# B&R Automation Studio project Riesenrad_Noecker
Automation Studio 4.9

## Configuration Config1

### Hardware
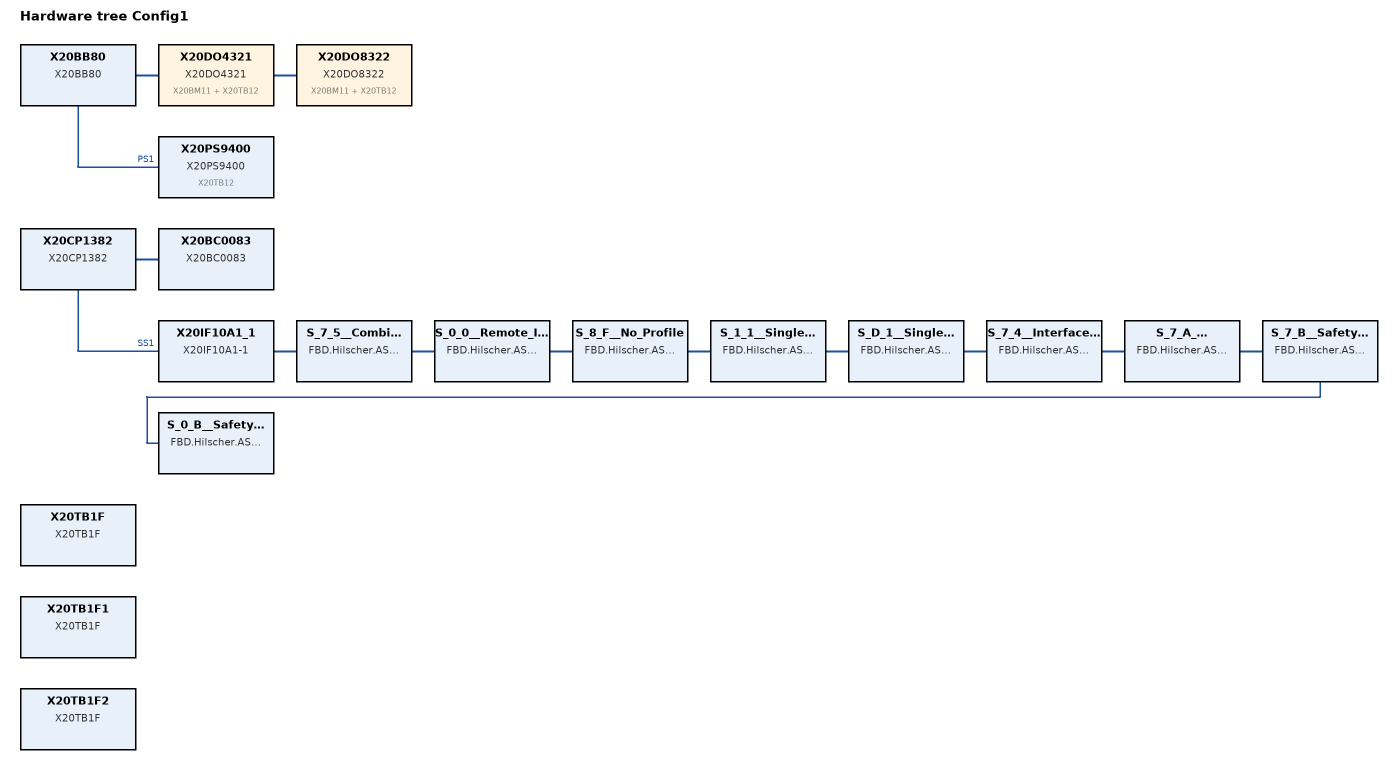
```
S_0_0__Remote_I_O_Port : FBD.Hilscher.AS-iSlaveDTM.S-0.0, Remote I$002FO Port vv.1 (OrderNumber=S-0.0, Remote I/O Port, VendorAddress=6)  [ASI1 -> S_7_5__Combi_field_device.ASI2]
  DtmId = cf450b26-e8ff-40bc-9c63-3c82782502b7
S_0_B__Safety_Slave : FBD.Hilscher.AS-iSlaveDTM.S-0.B, Safety Slave vv.1 (OrderNumber=S-0.B, Safety Slave, VendorAddress=13)  [ASI1 -> S_7_B__Safety_Slave.ASI2]
  DtmId = fa895fa4-d2e2-420c-b180-d2f2a02c2746
S_1_1__Single_Sensor__ext__contrl__ : FBD.Hilscher.AS-iSlaveDTM.S-1.1, Single Sensor (ext. contrl.) vv.1 (OrderNumber=S-1.1, Single Sensor (ext. contrl.), VendorAddress=8)  [ASI1 -> S_8_F__No_Profile.ASI2]
  DtmId = 9d5958e7-af56-4891-85b2-a17b108117c6
  ChannelBlocks_d3a35aad-8872-4e6a-914e-a881e2e31eaf  // Digital Input   [IN, 3 Bit(s)]
  ChannelBlocks_5bb377f7-42b1-4be2-805b-3354552dfad2  // Digital Output   [OUT, 1 Bit(s)]
S_7_4__Interface_for_16_bit_Signals : FBD.Hilscher.AS-iSlaveDTM.S-7.4, Interface for 16-bit Signals vv.1 (OrderNumber=S-7.4, Interface for 16-bit Signals, VendorAddress=10)  [ASI1 -> S_D_1__Single_Actuator_with_Monitoring.ASI2]
  DtmId = 0448b8e5-dced-4082-b80d-faf59c51bd2e
S_7_5__Combi_field_device : FBD.Hilscher.AS-iSlaveDTM.S-7.5, Combi field device vv.1 (OrderNumber=S-7.5, Combi field device, VendorAddress=5)  [ASI1 -> X20IF10A1_1.IF1]
  DtmId = 67ecf5d0-7b03-43bf-b517-437fc573c51f
S_7_A__Extended_Addressing_Mode : FBD.Hilscher.AS-iSlaveDTM.S-7.A, Extended Addressing Mode vv.1 (OrderNumber=S-7.A, Extended Addressing Mode, VendorAddress=11A)  [ASI1 -> S_7_4__Interface_for_16_bit_Signals.ASI2]
  DtmId = aa6d7d95-ba0b-4b78-a67e-6a7357710189
S_7_B__Safety_Slave : FBD.Hilscher.AS-iSlaveDTM.S-7.B, Safety Slave vv.1 (OrderNumber=S-7.B, Safety Slave, VendorAddress=12)  [ASI1 -> S_7_A__Extended_Addressing_Mode.ASI2]
  DtmId = 9a4111d3-a435-40ac-aa39-f4e884879d03
S_8_F__No_Profile : FBD.Hilscher.AS-iSlaveDTM.S-8.F, No Profile vv.1 (OrderNumber=S-8.F, No Profile, VendorAddress=7)  [ASI1 -> S_0_0__Remote_I_O_Port.ASI2]
  DtmId = 9c96085a-2bbf-4131-ae5e-8f64e9332ff0
S_D_1__Single_Actuator_with_Monitoring : FBD.Hilscher.AS-iSlaveDTM.S-D.1, Single Actuator with Monitoring vv.1 (OrderNumber=S-D.1, Single Actuator with Monitoring, VendorAddress=9)  [ASI1 -> S_1_1__Single_Sensor__ext__contrl__.ASI2]
  DtmId = 7ec07f93-a328-4a1d-a195-20a6fc18844a
  ChannelBlocks_4557325d-69fd-4a76-8f74-a661177b6065  // Digital Input   [IN, 3 Bit(s)]
  ChannelBlocks_a4a1c77a-8520-4756-9f44-c27872900355  // Digital Output   [OUT, 1 Bit(s)]
X20BB80 : X20BB80 v1.1.0.0
X20BC0083 : X20BC0083 v2.14.0.0  [PLK1 -> X20CP1382.IF3 (NodeNumber=1) [Cable Type=PowerlinkCable, Length=10, Version=1.0.0.3]; SL -> X20BB80.SL1]
X20BM11 : X20BM11 v1.1.0.0  [X2X1 -> X20BB80.IF1]
X20BM11a : X20BM11 v1.1.0.0  [X2X1 -> X20BM11.X2X2]
X20CP1382 : X20CP1382 v1.14.0.0  [X1 -> X1.SL; X2 -> X2.SL; X3 -> X3.SL]
  Module X1 (Type=X1, Virtual=true, Version=1.14.0.0)
    Connection (Connector=SS1, TargetModule=X20TB1F, TargetConnector=SS)
    Connection (Connector=SL, TargetModule=X20CP1382, TargetConnector=X1)
  Module X2 (Type=X2, Virtual=true, Version=1.14.0.0)
    Connection (Connector=SS1, TargetModule=X20TB1F1, TargetConnector=SS)
    Connection (Connector=SL, TargetModule=X20CP1382, TargetConnector=X2)
  Module X3 (Type=X3, Virtual=true, Version=1.14.0.0)
    Connection (Connector=SS1, TargetModule=X20TB1F2, TargetConnector=SS)
    Connection (Connector=SL, TargetModule=X20CP1382, TargetConnector=X3)
  Connector IF2:
    ActivateDevice = 1
    Mode = Manual
    InternetAddress = 192.168.0.10
    SubnetMask = 255.255.255.0
    ActivateSnmp = 2
  ConfigurationID = X20CP1382_Config1
  ActivateOpcUa = 1
  OpcUaInformationModels_PV_Version = 1
X20DO4321 : X20DO4321 v1.2.0.0  [SS1 -> X20TB12a.SS; SL -> X20BM11.SL1]
X20DO8322 : X20DO8322 v1.5.0.0  [SS1 -> X20TB12b.SS; SL -> X20BM11a.SL1]
X20IF10A1_1 : X20IF10A1-1 v1.3.0.0  [SS -> X20CP1382.SS1]
  Connector IF1:
    DtmId = c3d12960-2f64-4539-90e3-82e1d2b1aebe
  ConfigFile = X20IF10A1_1.dtm
  ConfigModule = asnxdb1
X20PS9400 : X20PS9400 v1.8.0.0  [SS1 -> X20TB12.SS; PS -> X20BB80.PS1]
X20TB12 : X20TB12 v1.0.0.0
X20TB12a : X20TB12 v1.0.0.0
X20TB12b : X20TB12 v1.0.0.0
X20TB1F : X20TB1F v1.0.0.0
X20TB1F1 : X20TB1F v1.0.0.0
X20TB1F2 : X20TB1F v1.0.0.0
```

### IoMap.iom - X20CP1382/IoMap.iom
```iecst
VAR_CONFIG
	::gDisplay AT %QW."S_7_5__Combi_field_device".Analog_Output_16_bit_Output_001;
	::gButtonOnOff AT %IX."S_0_0__Remote_I_O_Port".Digital_Input_1_bit_Input_001;
	::gButtonFast AT %IX."S_0_0__Remote_I_O_Port".Digital_Input_1_bit_Input_002;
	::gButtonSlow AT %IX."S_0_0__Remote_I_O_Port".Digital_Input_1_bit_Input_003;
	::gButtonStop AT %IX."S_0_0__Remote_I_O_Port".Digital_Input_1_bit_Input_004;
	::gRedDown AT %QX."S_8_F__No_Profile".Digital_Output_1_bit_Output_001;
	::gGreenDown AT %QX."S_8_F__No_Profile".Digital_Output_1_bit_Output_002;
	::gRedTop AT %QX."S_8_F__No_Profile".Digital_Output_1_bit_Output_003;
	::gGreenTop AT %QX."S_8_F__No_Profile".Digital_Output_1_bit_Output_004;
	::gReciever AT %IX."S_1_1__Single_Sensor__ext__contrl__".Digital_Input_1_bit_Input_001;
	::gTransmitter AT %QX."S_D_1__Single_Actuator_with_Monitoring".Digital_Output_1_bit_Output_001;
	::gRFIDColor AT %IW."S_7_4__Interface_for_16_bit_Signals".Analog_Input_16_bit_Input_001;
	::gASIStart AT %IX."S_7_A__Extended_Addressing_Mode".Digital_Input_1_bit_Input_001;
	::gASIStop AT %IX."S_7_A__Extended_Addressing_Mode".Digital_Input_1_bit_Input_002;
	::gASIQuit AT %IX."S_7_A__Extended_Addressing_Mode".Digital_Input_1_bit_Input_003;
	::gASISetup AT %IX."S_7_A__Extended_Addressing_Mode".Digital_Input_1_bit_Input_004;
	::gASILight1 AT %QX."S_7_A__Extended_Addressing_Mode".Digital_Output_1_bit_Output_001;
	::gASILight2 AT %QX."S_7_A__Extended_Addressing_Mode".Digital_Output_1_bit_Output_002;
	::gASILight3 AT %QX."S_7_A__Extended_Addressing_Mode".Digital_Output_1_bit_Output_003;
	::gEmergencyStop1 AT %IX."S_7_B__Safety_Slave".Digital_Input_1_bit_Input_001;
	::gEmergencyStop2 AT %IX."S_7_B__Safety_Slave".Digital_Input_1_bit_Input_002;
	::gEmergencyStop3 AT %IX."S_7_B__Safety_Slave".Digital_Input_1_bit_Input_003;
	::gEmergencyStop4 AT %IX."S_7_B__Safety_Slave".Digital_Input_1_bit_Input_004;
	::gLightGrid1 AT %IX."S_0_B__Safety_Slave".Digital_Input_1_bit_Input_001;
	::gLightGrid2 AT %IX."S_0_B__Safety_Slave".Digital_Input_1_bit_Input_002;
	::gLightGrid3 AT %IX."S_0_B__Safety_Slave".Digital_Input_1_bit_Input_003;
	::gLightGrid4 AT %IX."S_0_B__Safety_Slave".Digital_Input_1_bit_Input_004;
	::gDriveDirection AT %QX."X20DO4321".DigitalOutput01;
	::gDriveSpeed1 AT %QX."X20DO4321".DigitalOutput02;
	::gDriveSpeed2 AT %QX."X20DO4321".DigitalOutput03;
	::gSpotlightRight AT %QX."X20DO8322".DigitalOutput01;
	::gSpotlightLeft AT %QX."X20DO8322".DigitalOutput02;
	::gLightRed AT %QX."X20DO8322".DigitalOutput03;
	::gLightGreen AT %QX."X20DO8322".DigitalOutput04;
	::gLED1 AT %QX."X20DO8322".DigitalOutput05;
	::gLED2 AT %QX."X20DO8322".DigitalOutput06;
	::gLED3 AT %QX."X20DO8322".DigitalOutput07;
	::gLED4 AT %QX."X20DO8322".DigitalOutput08;
END_VAR
```

## Logical view

### Global.var - Globale Variablen
```iecst
(*List of global Variables*)
(* *)
VAR
	gSafetyStop : BOOL;
	gEmergencyStop : BOOL;
	gLightGrid : BOOL;
END_VAR
(*List of Variables for IO*)
(* *)
(*RFID*)
VAR
	gRFIDColor : UINT;
END_VAR
(* *)
(*Operating Light*)
VAR
	gRedTop : BOOL := FALSE;
	gGreenTop : BOOL := FALSE;
	gRedDown : BOOL := FALSE;
	gGreenDown : BOOL := FALSE;
END_VAR
(* *)
(*Drive*)
VAR
	gDriveDirection : BOOL := TRUE;
	gDriveSpeed1 : BOOL := FALSE;
	gDriveSpeed2 : BOOL := FALSE;
END_VAR
(* *)
(*Light*)
VAR
	gSpotlightRight : BOOL := FALSE;
	gSpotlightLeft : BOOL := FALSE;
	gLightRed : BOOL := TRUE;
	gLightGreen : BOOL := FALSE;
	gLED1 : BOOL := FALSE;
	gLED2 : BOOL := FALSE;
	gLED3 : BOOL := FALSE;
	gLED4 : BOOL := FALSE;
END_VAR
(* *)
(*Control Center*)
VAR
	gDisplay : UINT := 16#0505;
	gButtonOnOff : BOOL;
	gButtonFast : BOOL;
	gButtonSlow : BOOL;
	gButtonStop : BOOL;
END_VAR
(* *)
(*Light Barrier*)
VAR
	gReciever : BOOL;
	gTransmitter : BOOL := FALSE; (*For Activation on 1*)
END_VAR
(* *)
(*ASI Button*)
VAR
	gASIStart : BOOL;
	gASIStop : BOOL;
	gASIQuit : BOOL;
	gASISetup : BOOL;
	gASILight1 : BOOL := FALSE;
	gASILight2 : BOOL := FALSE;
	gASILight3 : BOOL := FALSE;
	gEmergencyStop1 : BOOL;
	gEmergencyStop2 : BOOL;
	gEmergencyStop3 : BOOL;
	gEmergencyStop4 : BOOL;
END_VAR
(* *)
(*Sicherheitsgitter*)
VAR
	gLightGrid1 : BOOL;
	gLightGrid2 : BOOL;
	gLightGrid3 : BOOL;
	gLightGrid4 : BOOL;
END_VAR
```

### Program Logical/Program (IEC)

#### Init.st - Init code
```iecst
PROGRAM _INIT
	(* Insert code here *)

	bSafetyResetReq:=TRUE;

	aPersonInCarSet[0]:=5;
	aPersonInCarSet[1]:=5;
	aPersonInCarSet[2]:=5;
	aPersonInCarSet[3]:=5;
	aPersonInCarSet[4]:=5;
	aPersonInCarSet[5]:=5;

	aRFIDColors[0]:=125; 	//red
	aRFIDColors[1]:=1280;	//pruple
	aRFIDColors[2]:=1536;	//white
	aRFIDColors[3]:=512;	//blue
	aRFIDColors[4]:=1024;	//yellow
	aRFIDColors[5]:=256;	//green

	bAutoMode:=TRUE;
	bSetup:=TRUE;
	gTransmitter:=TRUE;
	gASILight1:=FALSE;
	gASILight2:=FALSE;
	gASILight3:=FALSE;
	nLEDVisu:=0;
	nSpinnCountSet:=4;

	bAutomodeChange:=FALSE;
	bAutoMode:=FALSE;
	bModuloBusy:=FALSE;
END_PROGRAM
```

#### Types.typ - Local data types
```iecst
TYPE
	E_Speed :
		(
		fast := 2,
		slow := 1,
		stop := 0,
		normal := 3
		);
	E_AutoControl :
		(
		idle := 0,
		getout := 4,
		nextRFID := 2,
		spinn := 3,
		end := 5,
		getin := 1,
		nextRFIDout := 6
		);
END_TYPE
```

#### Drive.st
```iecst
ACTION Drive:
	CASE eSpeed OF
		stop:
			gDriveSpeed1:=0;
			gDriveSpeed2:=0;

		slow:
			gDriveSpeed1:=1;
			gDriveSpeed2:=0;

		fast:
			gDriveSpeed1:=1;
			gDriveSpeed2:=1;

		normal:
			gDriveSpeed1:=0;
			gDriveSpeed2:=1;

	END_CASE
END_ACTION
```

#### Display.st
```iecst
ACTION Display:
	IF NOT gSafetyStop AND NOT bSafetyResetReq THEN
		IF bAutoMode THEN
			sVisuMode:='Automatik';
			gDisplay:=16#0505;
			IF bSetup THEN
				sDisplayVisu:='Setup';
			ELSIF eAutoControl=idle THEN
				sDisplayVisu:='Fahre bis Rot';
			END_IF
			CASE eAutoControl OF
				getin:
					sDisplayVisu:='Einsteigen';
					gDisplay:=16#050C;

				getout:
					sDisplayVisu:='Aussteigen';
					gDisplay:=16#050C;

				spinn:
					sDisplayVisu:='Umlauf';
					gDisplay:=16#050E;

				nextRFID:
					sDisplayVisu:='Fahre zu nächster Gondel';
					gDisplay:=16#0505;

				nextRFIDout:
					sDisplayVisu:='Fahre zu nächster Gondel';
					gDisplay:=16#0505;
				end:
					sDisplayVisu:='Alle Gäste Ausgestiegen';
					gDisplay:=16#0505;

				idle:
					gDisplay:=16#0505;

			END_CASE

		ELSE
				sVisuMode:='Manual';
			CASE eSpeed OF
				stop:
					sDisplayVisu:='Keine Bewegung';
					gDisplay:=16#0A0B;

				slow:
					sDisplayVisu:='Langsam';
					gDisplay:=16#060B;

				fast:
					sDisplayVisu:='Schnell';
					gDisplay:=16#070B;
				normal:
					sDisplayVisu:='Normal';
						gDisplay:=16#050B;
			END_CASE

			IF bGondelsNotEmpty AND eSpeed = stop THEN
				sDisplayVisu:='Automatik nicht Möglich';
			END_IF
		END_IF
	ELSE
		sDisplayVisu:='Störung';
		gDisplay:=16#050A;

	END_IF

END_ACTION
```

#### Setup.st
```iecst
ACTION Setup:

	rSetup(CLK:=gASISetup);
	eAutoControl:=idle;
	IF rSetup.Q THEN
		gDriveDirection:=NOT gDriveDirection;

	ELSIF gASIStart THEN
		bSetup:=FALSE;
		bAutoMode:=TRUE;
	END_IF

	IF tonStart.Q THEN
		gASILight1:=NOT gASILight1;
	END_IF

	IF bSetAllGondels THEN
		aPersonInCarSet[0]:=nGondelValueSet;
		aPersonInCarSet[1]:=nGondelValueSet;
		aPersonInCarSet[2]:=nGondelValueSet;
		aPersonInCarSet[3]:=nGondelValueSet;
		aPersonInCarSet[4]:=nGondelValueSet;
		aPersonInCarSet[5]:=nGondelValueSet;
		bSetAllGondels:=FALSE;
	END_IF
	tonStart(IN:=(NOT tonStart.Q), PT:=T#1s);
END_ACTION
```

#### Automatic.st
```iecst
ACTION Automatic:
	gASILight1:=FALSE;
	CASE eAutoControl OF
		idle:
			eSpeed:=normal;
			IF gRFIDColor = aRFIDColors[0] THEN //Fahre bis Rot
				eSpeed:=stop;
				gLightGreen:=TRUE;
				RisingLightBarrier.CLK:=gReciever;
				eAutoControl:=getin;
				nLastRFIDAuto:=0;
				nSpinnCountIs:=0;
			END_IF

		getin:
			gLightGreen:=TRUE;
			gLightRed:=FALSE;
			IF RisingLightBarrier.Q THEN
				aPersonInCarIs[nRFIDArrIndex]:=aPersonInCarIs[nRFIDArrIndex]+1;
			END_IF

			IF aPersonInCarIs[nRFIDArrIndex]=aPersonInCarSet[nRFIDArrIndex] THEN
				IF (NOT gDriveDirection AND nRFIDArrIndex=1) OR ( gDriveDirection AND nRFIDArrIndex=5) THEN
					eAutoControl:=spinn;
				ELSE
					eAutoControl:=nextRFID;
					gLightGreen:=FALSE;
					gLightRed:=TRUE;
				END_IF

			END_IF

		nextRFID:
			gLightGreen:=FALSE;
			gLightRed:=TRUE;
			eSpeed:=slow;
			gLightGreen:=FALSE;
			gLightRed:=TRUE;
			IF gRFIDColor <> 0 AND gRFIDColor <> nLastRFIDAuto THEN
				eSpeed:=stop;
				nLastRFIDAuto:=gRFIDColor;
				gLightGreen:=TRUE;
				gTransmitter:=TRUE;
				bNextRFID:=FALSE;
				eAutoControl:=getin;
			END_IF

		spinn:
			gLightGreen:=FALSE;
			gLightRed:=TRUE;
			rRFIDTrack.CLK:=nLastRFID = aRFIDColors[0];
			eSpeed:=fast;
			bNextRFID:=FALSE;
			IF nSpinnCountIs = nSpinnCountSet THEN
				eSpeed:=normal;
				eAutoControl:=getout;
				nSpinnCountIs:=0;
			ELSIF rRFIDTrack.Q THEN
				nSpinnCountIs:=nSpinnCountIs+1;
			END_IF

		getout:
			eSpeed:=stop;
			gLightGreen:=FALSE;
			gLightRed:=TRUE;
			IF RisingLightBarrier.Q THEN
				aPersonInCarIs[nRFIDArrIndex]:=aPersonInCarIs[nRFIDArrIndex]-1;
			END_IF

			IF aPersonInCarIs[nRFIDArrIndex]=0 THEN
				IF (NOT gDriveDirection AND nRFIDArrIndex=1) OR (gDriveDirection AND nRFIDArrIndex=5) THEN
					eAutoControl:=end;
				ELSE
					eAutoControl:=nextRFIDout;
					gLightGreen:=FALSE;
					gLightRed:=TRUE;
				END_IF

			END_IF

		nextRFIDout:
			gLightGreen:=FALSE;
			gLightRed:=TRUE;

				eSpeed:=slow;
				gLightGreen:=FALSE;
				gLightRed:=TRUE;
			IF gRFIDColor <> 0 AND  gRFIDColor <> nLastRFIDAuto THEN
				nLastRFIDAuto:=gRFIDColor;
					eSpeed:=stop;
					gLightGreen:=TRUE;
					gTransmitter:=TRUE;
					eAutoControl:=getout;
					bNextRFID:=FALSE;

				END_IF
		end:
			gASILight1:=TRUE;
			rAsiStart.CLK:=gASIStart;
			IF rAsiStart.Q THEN
				tonTimerRun.IN:=TRUE;
			END_IF

			IF tonTimerRun.Q AND NOT gASIStart THEN
				tonTimerRun.IN:=FALSE;
				bSetup:=TRUE;
				gASILight1:=FALSE;
				eAutoControl:=idle;

			END_IF

	END_CASE
	RisingLightBarrier.CLK:=gReciever;
	RisingLightBarrier();
	tonTimerRun(PT:=T#500ms);
	rSetup();
	rRFIDTrack();
	rAsiStart();
END_ACTION
```

#### Visu.st
```iecst
ACTION Visu:

	FOR i:=0 TO 5 DO
		aVisuRFIDCol[i]:=0;
	END_FOR
	IF gRFIDColor <> 0 THEN
		nLastRFID:=gRFIDColor;

	END_IF

	CASE nLastRFID OF
		125:
			nCurrentPerson:=aPersonInCarIs[0];
			aVisuRFIDCol[0]:=TRUE;
			nRFIDArrIndex:=0;

		512:
			nCurrentPerson:=aPersonInCarIs[3];
			aVisuRFIDCol[3]:=TRUE;
			nRFIDArrIndex:=3;
		256:
			nCurrentPerson:=aPersonInCarIs[5];
			aVisuRFIDCol[5]:=TRUE;
			nRFIDArrIndex:=5;
		1536:
			nCurrentPerson:=aPersonInCarIs[2];
			aVisuRFIDCol[2]:=TRUE;
			nRFIDArrIndex:=2;
		1280:
			nCurrentPerson:=aPersonInCarIs[1];
			aVisuRFIDCol[1]:=TRUE;
			nRFIDArrIndex:=1;
		1024:
			nCurrentPerson:=aPersonInCarIs[4];
			aVisuRFIDCol[4]:=TRUE;
		nRFIDArrIndex:=4;
	END_CASE

	IF bSetup AND gDriveDirection THEN
		sVisuDrehrichtung:='gegen Uhr';
	ELSIF bSetup AND NOT gDriveDirection THEN
		sVisuDrehrichtung:='mit Uhr';
	END_IF

END_ACTION
```

- Visualisation Logical/mappView (not shown)

Listed in the project but not available here: Logical/Global.typ, Logical/Libraries, Logical/Program/Cyclic.st, Logical/Program/Exit.st, Logical/Program/Variables.var, Logical/Program/Safety.st, Logical/Program/Manual.st, Logical/Program/Lights.st
